// TIA Portal V20 export
ORGANIZATION_BLOCK "Startup"   // OB100, FBD, Startup
TITLE = "Complete Restart"
{ S7_Optimized_Access := 'TRUE' }
// stored: SetENOAutomatically false
   VAR_INPUT
      LostRetentive : Bool;   // True if retentive data are lost
      LostRTC : Bool;   // True if date and time are lost
   END_VAR
BEGIN

NETWORK
TITLE = first scan
      SET;
      S     "firstScan";

NETWORK
TITLE = call diagnose
      CALL  "Diag", "Diag_DB";

END_ORGANIZATION_BLOCK
